(* Verify that the statuses of the switchbox valves match the expected statuses *)
FUNCTION F_VerifySBValveStatuses : BOOL
VAR_INPUT
	stExpStatus : ST_SBValveStatuses; // The expected state of the system
	bEnforce : BOOL; // Whether to try forcing the states
END_VAR
VAR
	stStatus : ST_SBValveStatuses;
END_VAR

stStatus := F_GetSBValveStatuses();

IF bEnforce THEN
	// Try setting system states to the expected states
	F_SetSBValveStatuses(stExpStatus);
END_IF

// Return true if the expected status matches the actual status
F_VerifySBValveStatuses := stExpStatus.bGateValveOpen = stStatus.bGateValveOpen
	AND stExpStatus.bVentValveOpen = stStatus.bVentValveOpen
	AND stExpStatus.bORingPumpValveOpen = stStatus.bORingPumpValveOpen
	AND stExpStatus.bForelineValveOpen = stStatus.bForelineValveOpen
	AND stExpStatus.bSBVentOpen = stStatus.bSBVentOpen
	AND stExpStatus.bSlowPumpValveOpen = stStatus.bSlowPumpValveOpen
	AND stExpStatus.bSBSlowVentOpen = stStatus.bSBSlowVentOpen;

END_FUNCTION

(* stored: Version 1.1.0.1, ProductVersion 3.1.4024.0
   POU F_VerifySBValveStatuses: Id {7e9e080f-6367-40a9-93e1-9bb54b843059}, SpecialFunc None *)
